// TwinCAT 3 PLC project CarRep_1120_Sagedergasse
// ProgramVersion: 3.1.4023.0
// libraries:
//   Lynus Energy Basic, * (Lynus AG)
//   Lynus Energy ModbusTCP, * (Lynus AG)
//   Lynus Standards, * (Lynus AG)
//   Tc2_ModbusSrv, * (Beckhoff Automation GmbH)
//   Tc2_Standard, * (Beckhoff Automation GmbH)
//   Tc2_System, * (Beckhoff Automation GmbH)
//   Tc3_Module, * (Beckhoff Automation GmbH)
//   TSG Communicator, * (EfficientIO)
// project tree:
//   / FastTask.TcTTO, MiddleTask.TcTTO, SlowTask.TcTTO
//   POUs/ prgComTSG.TcPOU, prgCS.TcPOU, prgEMS.TcPOU, prgRWTSG.TcPOU, prgVarTSG.TcPOU
// real-time tasks:
//   TASK FastTask: cycle T#5ms, priority 6, ADS port 350
//   TASK MiddleTask: cycle T#10ms, priority 8, ADS port 351
//   TASK SlowTask: cycle T#20ms, priority 10, ADS port 352

CONFIGURATION CarRep_1120_Sagedergasse
    RESOURCE PLC ON TwinCAT3
        TASK FastTask(INTERVAL := T#5ms, PRIORITY := 6);
        TASK MiddleTask(INTERVAL := T#10ms, PRIORITY := 8);
        TASK SlowTask(INTERVAL := T#20ms, PRIORITY := 10);
        PROGRAM prgRWTSG WITH FastTask : prgRWTSG;
        PROGRAM prgVarTSG WITH FastTask : prgVarTSG;
        PROGRAM prgCS WITH MiddleTask : prgCS;
        PROGRAM prgEMS WITH MiddleTask : prgEMS;
        PROGRAM prgComTSG WITH SlowTask : prgComTSG;
    END_RESOURCE
END_CONFIGURATION

// ---- POUs/prgRWTSG.TcPOU
PROGRAM prgRWTSG
VAR
	fbRW1		: FB_ReadWrite;
END_VAR

fbRW1(bBusy=> , bError=> , udiErrorCodeOut=> , eErrorReadWrite_Out=> );

END_PROGRAM

// ---- POUs/prgVarTSG.TcPOU
PROGRAM prgVarTSG
VAR
	fbVar		: FB_VarInfo;
END_VAR

fbVar(
	bReadInfo:= , 
	eTMCFile:= eSelectTMCFile.eDontUseTMCFile, 
	eSavePositionTMCFile:= eSavePositionOnPLC.ePostionHardDisk, 
	udiCounterFoundVariables=> , 
	bError=> , 
	bBusy=> , 
	byProgress=> , 
	udiErrorCodeOut=> , 
	eErrorVarInfo_Out=> , 
	sVarWithError=> );

END_PROGRAM

// ---- POUs/prgCS.TcPOU
PROGRAM prgCS
VAR
	fbAlfen1					: FB_ECS_Alfen_NG9xx_Platform;						//{#lynus.ag#()}
	fbAlfen2					: FB_ECS_Alfen_NG9xx_Platform;						//{#lynus.ag#()}
	bSManualyOnCS1				: BOOL;												//{#lynus.ag#()}
	bySManualyTargetPowerCS1	: BYTE;												//{#lynus.ag#()}
	byErrorWarningCS1			: BYTE;												//{#lynus.ag#()}
	bSManualyOnCS2				: BOOL;												//{#lynus.ag#()}
	bySManualyTargetPowerCS2	: BYTE;												//{#lynus.ag#()}
	byErrorWarningCS2			: BYTE;												//{#lynus.ag#()}
END_VAR
VAR PERSISTENT
	bManualyOnCS1				: BOOL;												//{#lynus.ag#()}
	byManualyTargetPowerCS1		: BYTE;												//{#lynus.ag#()}
	bManualyOnCS2				: BOOL;												//{#lynus.ag#()}
	byManualyTargetPowerCS2		: BYTE;												//{#lynus.ag#()}
END_VAR

//CS1 - EV DMU50120

//Manual Power
fbAlfen1.stSetupECS.bManualyOn := bManualyOnCS1;
	fbAlfen1.stSetupECS.byManualyTargetPower := byManualyTargetPowerCS1;

fbAlfen1(
	bEnable:= TRUE, 
	bPowerDataInvers:= , 
	byElectricFuseLine:= , 
	byUnitID_Socket1:= 1, 
	byUnitID_Socket2:= , 
	byNumberOfSockets:= 1, 
	byNumberOfConnectionWire:= 1, 
	diNrOfEMS_IN:= , 
	diNrOfEM_IN_CS:= , 
	sIPAdress:= '192.168.0.3', 
	stSetupECS:= , 
	stDataECS=> , 
	diNrOfECS_OUT=> );

bSManualyOnCS1 := fbAlfen1.stDataECS.bSManualyOn;
	bySManualyTargetPowerCS1 := fbAlfen1.stDataECS.bySManualyTargetPower;
		byErrorWarningCS1 := fbAlfen1.stDataECS.byErrorWarning;


//CS2 - EV DMU50089

//Manual Power
fbAlfen2.stSetupECS.bManualyOn := bManualyOnCS2;
	fbAlfen2.stSetupECS.byManualyTargetPower := byManualyTargetPowerCS2;

fbAlfen2(
	bEnable:= TRUE, 
	bPowerDataInvers:= , 
	byElectricFuseLine:= , 
	byUnitID_Socket1:= 1, 
	byUnitID_Socket2:= , 
	byNumberOfSockets:= 1, 
	byNumberOfConnectionWire:= 1, 
	diNrOfEMS_IN:= , 
	diNrOfEM_IN_CS:= , 
	sIPAdress:= '192.168.0.4', 
	stSetupECS:= , 
	stDataECS=> , 
	diNrOfECS_OUT=> );

bSManualyOnCS2 := fbAlfen2.stDataECS.bSManualyOn;
	bySManualyTargetPowerCS2 := fbAlfen2.stDataECS.bySManualyTargetPower;
		byErrorWarningCS2 := fbAlfen2.stDataECS.byErrorWarning;

END_PROGRAM

// ---- POUs/prgEMS.TcPOU
PROGRAM prgEMS
VAR
	fbEMS		: FB_EMS_V2;		//{#lynus.ag#()}
END_VAR

fbEMS(
	bEnable:= , 
	tDelayPwrCorrectionECS:= , 
	stNrOfEM_IN_ECS:= , 
	stSizeMainFuseCS:= , 
	stSetupEMS:= , 
	eOperationMode:= , 
	eSpeedModeBackendController:= E_SpeedModeBackendController_EMS.eSlow, 
	eSpeedModeLocalController:= E_SpeedModeLocalController_EMS.eSlow, 
	bActivateHP:= , 
	bControllingState:= , 
	rHeartbeat:= , 
	rErrorWarning:= , 
	rEnergyOptReady:= , 
	rNewBattPower:= , 
	eMessageEMS=> , 
	bStateEnable=> , 
	bStateAllowChrgFromGrid=> , 
	bMissingPowerData=> , 
	bSurplusAvailable=> , 
	bSEnableMainFuseFunc=> , 
	byProgress=> , 
	uiState_OUT=> , 
	diNrOfEMS_OUT=> , 
	arrMinPrioReached=> , 
	arrMaxPrioReached=> );

END_PROGRAM

// ---- POUs/prgComTSG.TcPOU
PROGRAM prgComTSG
VAR
	fbCom		: FB_MqttCommunicator;
END_VAR

fbCom(
	bConnect:= TRUE, 
	sUserName:= '806b5b3a-69a5-452f-af78-4b065bd4b761', 
	sUserPassword:= 'fbc367e6-1894-4e5e-8737-325595087c51', 
	eSavePositionCertificate:= eSavePositionOnPLC.ePostionHardDisk, 
	bConnected=> , 
	bError=> , 
	hrErrorCode=> , 
	eConnectionState=> , 
	eErrorMessage_Out=> );

END_PROGRAM
